// TIA Portal V17 export
// export: Created 2025-03-07T09:18:55.6310354Z, ExportSetting WithDefaults, DisplayName Totally Integrated Automation Portal, DisplayVersion V17 Update 8, DisplayName TIA Portal Openness, DisplayVersion V17 Update 8, DisplayName TIA Portal Version Control Interface, DisplayVersion V17, DisplayName SINAMICS Startdrive Advanced, DisplayVersion V17 SP2, DisplayName SINAMICS Startdrive G110M, G120, G120C, G120D, G120P, G115D, DisplayVersion V17 SP2, DisplayName SINAMICS Startdrive G130, G150, S120, S150, SINAMICS MV, S210, DisplayVersion V17 SP2, DisplayName STEP 7 Professional, DisplayVersion V17 Update 8, DisplayName SINUMERIK ONE STEP 7 Toolbox, DisplayVersion V17 Update 12, DisplayName SINUMERIK 840D sl STEP 7 Toolbox, DisplayVersion V17 Update 12, DisplayName STEP 7 Safety, DisplayVersion V17 Update 6, DisplayName WinCC Advanced, DisplayVersion V17 Update 8
DATA_BLOCK "DB20200_GENERAL_LASER"   // DB20200
{ S7_Optimized_Access := 'TRUE'; DB_Accessible_From_OPC_UA := 'FALSE' }
VERSION : 0.1
// stored: AutoNumber false, DBAccessibleFromOPCUA false, DBAccessibleFromWebserver true, IsOnlyStoredInLoadMemory false, IsRetainMemResEnabled false, IsWriteProtectedInAS false, MemoryReserve 100
   VAR
      "ALL LASERS READY" : Bool;
      "ALL LASERS UNIT 1 READY" : Bool;
      "ALL LASERS UNIT 2 READY" : Bool;
      AXIS_U01_NOT_MOVE_FAULT : Bool;   // AXIS FROM UNIT 01 NOT MOVING WHILE LASER ON FAULT
      AXIS_U02_NOT_MOVE_FAULT : Bool;   // AXIS FROM UNIT 01 NOT MOVING WHILE LASER ON FAULT
      AXIS_U01_NOT_MOVE_FAULT_TIMER : IEC_TIMER;   // AXIS FROM UNIT 01 NOT MOVING WHILE LASER ON FAULT TIMER
      AXIS_U02_NOT_MOVE_FAULT_TIMER : IEC_TIMER;   // AXIS FROM UNIT 02 NOT MOVING WHILE LASER ON FAULT TIMER
   END_VAR
BEGIN
END_DATA_BLOCK
